// TIA Portal V16 export
// export: Created 2024-05-10T06:46:43.0449817Z, ExportSetting WithDefaults, DisplayName Totally Integrated Automation Portal, DisplayVersion V16, DisplayName TIA Portal Version Control Interface, DisplayVersion V16, DisplayName TIA Portal Openness, DisplayVersion V16, DisplayName STEP 7 Professional, DisplayVersion V16, DisplayName STEP 7 Safety, DisplayVersion V16, DisplayName WinCC Professional, DisplayVersion V16
FUNCTION_BLOCK "F120_SinaPos(SV660F)"   // FB120, LAD
{ S7_Optimized_Access := 'TRUE' }
VERSION : 0.1
// 2024/2/4:第一版本V1.0，作者:wang
// stored: AutoNumber false, IsIECCheckEnabled false, IsRetainMemResEnabled false, MemoryReserve 100, SetENOAutomatically false, UDAEnableTagReadback false
   VAR_INPUT
      IW_手动模式 { ExternalAccessible := 'False'; ExternalVisible := 'False'; ExternalWritable := 'False'} : Bool;
      IW_运行条件 { ExternalAccessible := 'False'; ExternalVisible := 'False'; ExternalWritable := 'False'} : Array[1..8] of Bool;
      IM_使能 { ExternalAccessible := 'False'; ExternalVisible := 'False'; ExternalWritable := 'False'} : Bool;
      IM_回零 { ExternalAccessible := 'False'; ExternalVisible := 'False'; ExternalWritable := 'False'} : Bool;
      IM_绝对定位 { ExternalAccessible := 'False'; ExternalVisible := 'False'; ExternalWritable := 'False'} : Bool;
      IM_相对定位 { ExternalAccessible := 'False'; ExternalVisible := 'False'; ExternalWritable := 'False'} : Bool;
      "IM_JOG+" { ExternalAccessible := 'False'; ExternalVisible := 'False'; ExternalWritable := 'False'} : Bool;
      "IM_JOG-" { ExternalAccessible := 'False'; ExternalVisible := 'False'; ExternalWritable := 'False'} : Bool;
      IM_故障复位 { ExternalAccessible := 'False'; ExternalVisible := 'False'; ExternalWritable := 'False'} : Bool;
      ID_目标位置 { ExternalAccessible := 'False'; ExternalVisible := 'False'; ExternalWritable := 'False'} : DInt;
      ID_目标速度 { ExternalAccessible := 'False'; ExternalVisible := 'False'; ExternalWritable := 'False'} : DInt;
      "IW_速度加减倍率%" { ExternalAccessible := 'False'; ExternalVisible := 'False'; ExternalWritable := 'False'} : Array[1..3] of Int;
      ID_ConfigEpos { ExternalAccessible := 'False'; ExternalVisible := 'False'; ExternalWritable := 'False'} : DWord;
      ID_111报文标识符 { ExternalAccessible := 'False'; ExternalVisible := 'False'; ExternalWritable := 'False'} : HW_IO;
   END_VAR
   VAR_OUTPUT
      OM_准备好了 : Bool;
      OM_动作中 : Bool;
      OM_回零完了 : Bool;
      OM_轴报警 : Bool;
      OM_轴错误 : Bool;
      OD_当前位置 : DInt;
      OD_当前速度 : DInt;
      OW_运行模式 : Int;
      OW_EPSW1 : Word;
      OW_EPSW2 : Word;
      OW_轴报警码 : Word;
      OW_轴错误码 : Word;
      OW_库错误码 : Int;
      OW_调用错误码 : Word;
   END_VAR
   VAR
      MT_StartChk : IEC_TIMER;   // 启动延迟
   END_VAR
   VAR_TEMP
      M_停止 : Bool;
      M_暂停 : Bool;
      M_JOG指令 : Bool;
      M_回零指令 : Bool;
      M_绝对定位指令 : Bool;
      M_相对定位指令 : Bool;
      M_回零定位完Pls : Bool;
      M_绝对定位完Pls : Bool;
      M_相对定位完Pls : Bool;
      M_启动 : Bool;
      M_定位完了 : Bool;
      W_运行模式 : Int;
      M_Pulse : Array[1..20] of Bool;
      M_SerState : Bool;   // 伺服正常
      M_Busy : Bool;   // 伺服忙
      M_FLS_SW : Bool;   // 正极限
      M_RLS_SW : Bool;   // 负极限
   END_VAR
   // // IW_运行条件[1] : 共同条件
   // // IW_运行条件[2] : 回零条件
   // // IW_运行条件[3] : JOG正条件
   // // IW_运行条件[4] : JOG负条件
   // // IW_运行条件[5] : 定位正条件
   // // IW_运行条件[6] : 定位负条件
   // // IW_运行条件[7] : 预留
   // // IW_运行条件[8] : 预留
   VAR_TEMP   // added for the SCL form of the ladder/FBD networks
      _w1 : Bool;
      _w2 : Bool;
      _w3 : Bool;
      _w4 : Bool;
   END_VAR
BEGIN

REGION Network 1: 伺服状态条件
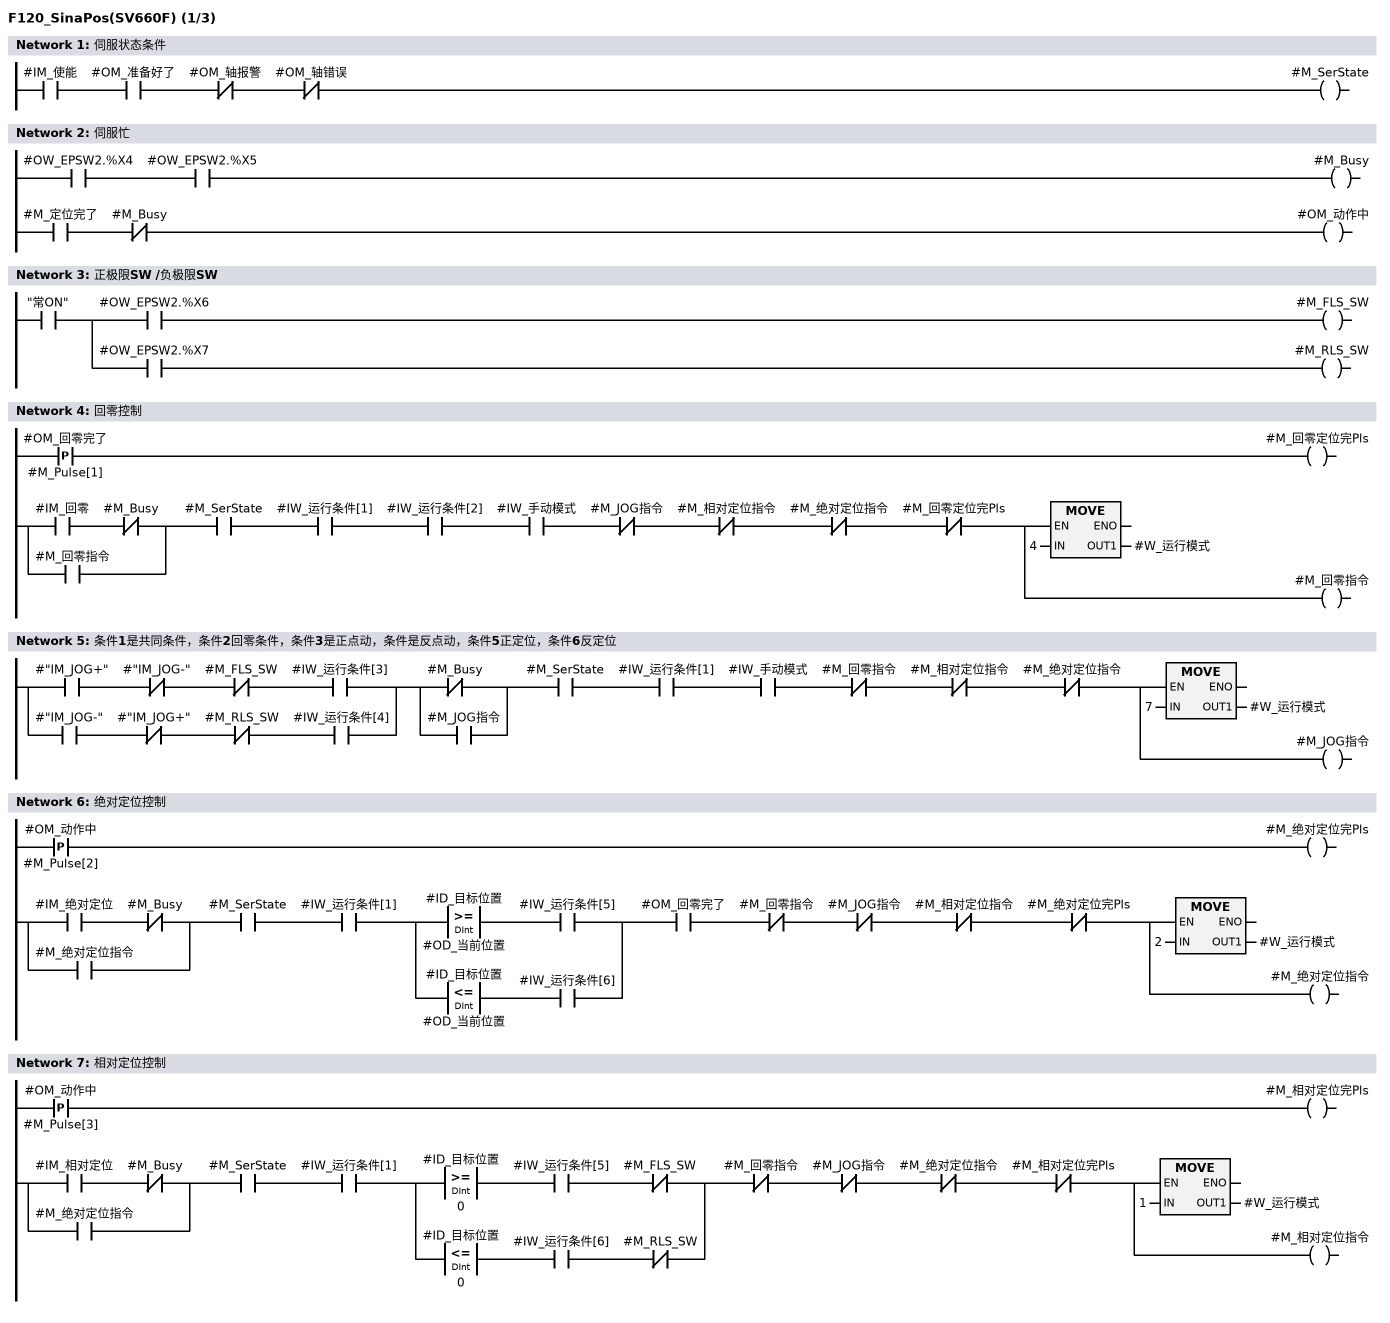
   RUNG wire#powerrail
      Contact( #IM_使能 )
      Contact( #OM_准备好了 )
      I_Contact( #OM_轴报警 )
      I_Contact( #OM_轴错误 )
      Coil( #M_SerState )
   END_RUNG
   // the same network as SCL:
   #M_SerState := #IM_使能 AND #OM_准备好了 AND NOT #OM_轴报警 AND NOT #OM_轴错误;
END_REGION

REGION Network 2: 伺服忙
   RUNG wire#powerrail
      Contact( #OW_EPSW2.%X4 )
      Contact( #OW_EPSW2.%X5 )
      Coil( #M_Busy )
   END_RUNG
   RUNG wire#powerrail
      Contact( #M_定位完了 )
      I_Contact( #M_Busy )
      Coil( #OM_动作中 )
   END_RUNG
   // the same network as SCL:
   #M_Busy := #OW_EPSW2.%X4 AND #OW_EPSW2.%X5;
   #OM_动作中 := #M_定位完了 AND NOT #M_Busy;
END_REGION

REGION Network 3: 正极限SW /负极限SW
   RUNG wire#powerrail
      Contact( "常ON" )
      wire#w1
      Contact( #OW_EPSW2.%X6 )
      Coil( #M_FLS_SW )
   END_RUNG
   RUNG wire#w1
      Contact( #OW_EPSW2.%X7 )
      Coil( #M_RLS_SW )
   END_RUNG
   // the same network as SCL:
   #M_FLS_SW := "常ON" AND #OW_EPSW2.%X6;
   #M_RLS_SW := "常ON" AND #OW_EPSW2.%X7;
END_REGION

REGION Network 4: 回零控制
   RUNG wire#powerrail
      P_Contact(operand := #OM_回零完了, bit := #M_Pulse[1])
      Coil( #M_回零定位完Pls )
   END_RUNG
   RUNG wire#powerrail
      Contact( #IM_回零 )
      I_Contact( #M_Busy )
      wire#w1
      Contact( #M_SerState )
      Contact( #IW_运行条件[1] )
      Contact( #IW_运行条件[2] )
      Contact( #IW_手动模式 )
      I_Contact( #M_JOG指令 )
      I_Contact( #M_相对定位指令 )
      I_Contact( #M_绝对定位指令 )
      I_Contact( #M_回零定位完Pls )
      wire#w2
      Move(in := 4, out1 => #W_运行模式)
   END_RUNG
   RUNG wire#powerrail
      Contact( #M_回零指令 )
   END_RUNG wire#w1
   RUNG wire#w2
      Coil( #M_回零指令 )
   END_RUNG
   // the same network as SCL:
   #_w1 := #OM_回零完了 AND NOT #M_Pulse[1];   // rising edge of #OM_回零完了
   #M_Pulse[1] := #OM_回零完了;
   #M_回零定位完Pls := #_w1;
   #_w2 := ((#IM_回零 AND NOT #M_Busy) OR #M_回零指令) AND #M_SerState AND #IW_运行条件[1] AND #IW_运行条件[2] AND #IW_手动模式 AND NOT #M_JOG指令 AND NOT #M_相对定位指令 AND NOT #M_绝对定位指令 AND NOT #M_回零定位完Pls;
   IF #_w2 THEN #W_运行模式 := 4; END_IF;
   #M_回零指令 := #_w2;
END_REGION

REGION Network 5: 条件1是共同条件，条件2回零条件，条件3是正点动，条件是反点动，条件5正定位，条件6反定位
   RUNG wire#powerrail
      Contact( #"IM_JOG+" )
      I_Contact( #"IM_JOG-" )
      I_Contact( #M_FLS_SW )
      Contact( #IW_运行条件[3] )
      wire#w1
      I_Contact( #M_Busy )
      wire#w2
      Contact( #M_SerState )
      Contact( #IW_运行条件[1] )
      Contact( #IW_手动模式 )
      I_Contact( #M_回零指令 )
      I_Contact( #M_相对定位指令 )
      I_Contact( #M_绝对定位指令 )
      wire#w3
      Move(in := 7, out1 => #W_运行模式)
   END_RUNG
   RUNG wire#powerrail
      Contact( #"IM_JOG-" )
      I_Contact( #"IM_JOG+" )
      I_Contact( #M_RLS_SW )
      Contact( #IW_运行条件[4] )
   END_RUNG wire#w1
   RUNG wire#w1
      Contact( #M_JOG指令 )
   END_RUNG wire#w2
   RUNG wire#w3
      Coil( #M_JOG指令 )
   END_RUNG
   // the same network as SCL:
   #_w1 := ((#"IM_JOG+" AND NOT #"IM_JOG-" AND NOT #M_FLS_SW AND #IW_运行条件[3]) OR (#"IM_JOG-" AND NOT #"IM_JOG+" AND NOT #M_RLS_SW AND #IW_运行条件[4])) AND (NOT #M_Busy OR #M_JOG指令) AND #M_SerState AND #IW_运行条件[1] AND #IW_手动模式 AND NOT #M_回零指令 AND NOT #M_相对定位指令 AND NOT #M_绝对定位指令;
   IF #_w1 THEN #W_运行模式 := 7; END_IF;
   #M_JOG指令 := #_w1;
END_REGION

REGION Network 6: 绝对定位控制
   RUNG wire#powerrail
      P_Contact(operand := #OM_动作中, bit := #M_Pulse[2])
      Coil( #M_绝对定位完Pls )
   END_RUNG
   RUNG wire#powerrail
      Contact( #IM_绝对定位 )
      I_Contact( #M_Busy )
      wire#w1
      Contact( #M_SerState )
      Contact( #IW_运行条件[1] )
      wire#w2
      { S7_Templates := "SrcType := DInt" } GE_Contact(in1 := #ID_目标位置, in2 := #OD_当前位置)
      Contact( #IW_运行条件[5] )
      wire#w3
      Contact( #OM_回零完了 )
      I_Contact( #M_回零指令 )
      I_Contact( #M_JOG指令 )
      I_Contact( #M_相对定位指令 )
      I_Contact( #M_绝对定位完Pls )
      wire#w4
      Move(in := 2, out1 => #W_运行模式)
   END_RUNG
   RUNG wire#powerrail
      Contact( #M_绝对定位指令 )
   END_RUNG wire#w1
   RUNG wire#w2
      { S7_Templates := "SrcType := DInt" } LE_Contact(in1 := #ID_目标位置, in2 := #OD_当前位置)
      Contact( #IW_运行条件[6] )
   END_RUNG wire#w3
   RUNG wire#w4
      Coil( #M_绝对定位指令 )
   END_RUNG
   // the same network as SCL:
   #_w1 := #OM_动作中 AND NOT #M_Pulse[2];   // rising edge of #OM_动作中
   #M_Pulse[2] := #OM_动作中;
   #M_绝对定位完Pls := #_w1;
   #_w2 := ((#IM_绝对定位 AND NOT #M_Busy) OR #M_绝对定位指令) AND #M_SerState AND #IW_运行条件[1] AND (((#ID_目标位置 >= #OD_当前位置) AND #IW_运行条件[5]) OR ((#ID_目标位置 <= #OD_当前位置) AND #IW_运行条件[6])) AND #OM_回零完了 AND NOT #M_回零指令 AND NOT #M_JOG指令 AND NOT #M_相对定位指令 AND NOT #M_绝对定位完Pls;
   IF #_w2 THEN #W_运行模式 := 2; END_IF;
   #M_绝对定位指令 := #_w2;
END_REGION

REGION Network 7: 相对定位控制
   RUNG wire#powerrail
      P_Contact(operand := #OM_动作中, bit := #M_Pulse[3])
      Coil( #M_相对定位完Pls )
   END_RUNG
   RUNG wire#powerrail
      Contact( #IM_相对定位 )
      I_Contact( #M_Busy )
      wire#w1
      Contact( #M_SerState )
      Contact( #IW_运行条件[1] )
      wire#w2
      { S7_Templates := "SrcType := DInt" } GE_Contact(in1 := #ID_目标位置, in2 := 0)
      Contact( #IW_运行条件[5] )
      I_Contact( #M_FLS_SW )
      wire#w3
      I_Contact( #M_回零指令 )
      I_Contact( #M_JOG指令 )
      I_Contact( #M_绝对定位指令 )
      I_Contact( #M_相对定位完Pls )
      wire#w4
      Move(in := 1, out1 => #W_运行模式)
   END_RUNG
   RUNG wire#powerrail
      Contact( #M_绝对定位指令 )
   END_RUNG wire#w1
   RUNG wire#w2
      { S7_Templates := "SrcType := DInt" } LE_Contact(in1 := #ID_目标位置, in2 := 0)
      Contact( #IW_运行条件[6] )
      I_Contact( #M_RLS_SW )
   END_RUNG wire#w3
   RUNG wire#w4
      Coil( #M_相对定位指令 )
   END_RUNG
   // the same network as SCL:
   #_w1 := #OM_动作中 AND NOT #M_Pulse[3];   // rising edge of #OM_动作中
   #M_Pulse[3] := #OM_动作中;
   #M_相对定位完Pls := #_w1;
   #_w2 := ((#IM_相对定位 AND NOT #M_Busy) OR #M_绝对定位指令) AND #M_SerState AND #IW_运行条件[1] AND (((#ID_目标位置 >= 0) AND #IW_运行条件[5] AND NOT #M_FLS_SW) OR ((#ID_目标位置 <= 0) AND #IW_运行条件[6] AND NOT #M_RLS_SW)) AND NOT #M_回零指令 AND NOT #M_JOG指令 AND NOT #M_绝对定位指令 AND NOT #M_相对定位完Pls;
   IF #_w2 THEN #W_运行模式 := 1; END_IF;
   #M_相对定位指令 := #_w2;
END_REGION

REGION Network 8: 控制启动
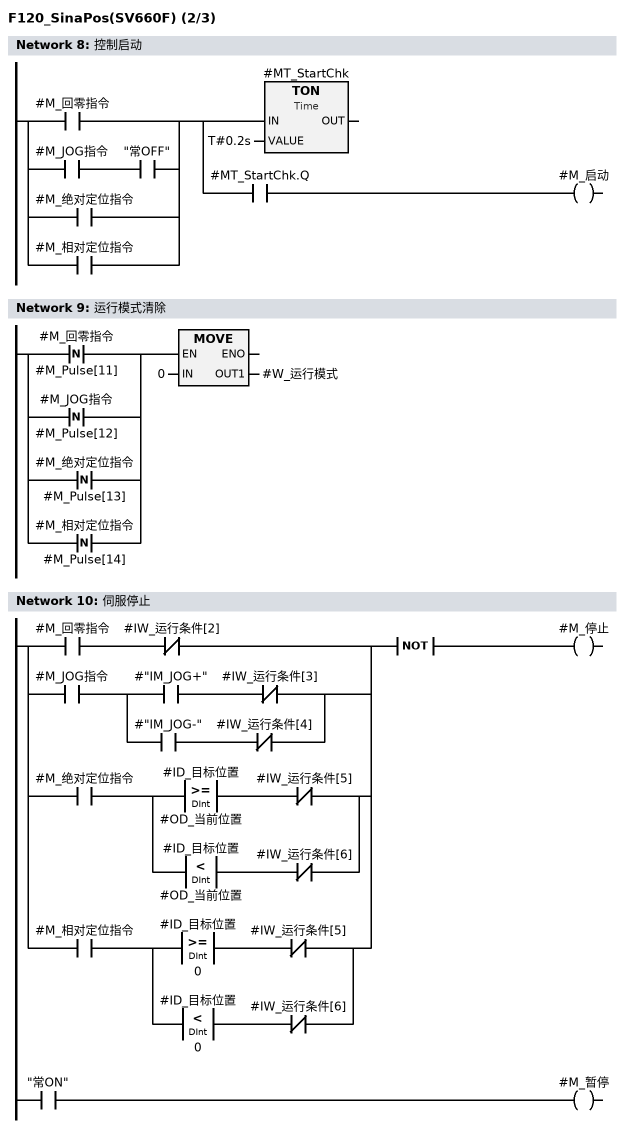
   #_w1 := #M_回零指令 OR (#M_JOG指令 AND "常OFF") OR #M_绝对定位指令 OR #M_相对定位指令;
   #MT_StartChk.TON(IN := #_w1, PT := T#0.2s);   // TON coil
   #M_启动 := #_w1 AND #MT_StartChk.Q;
END_REGION

REGION Network 9: 运行模式清除
   RUNG wire#powerrail
      N_Contact(operand := #M_回零指令, bit := #M_Pulse[11])
      wire#w1
      Move(in := 0, out1 => #W_运行模式)
   END_RUNG
   RUNG wire#powerrail
      N_Contact(operand := #M_JOG指令, bit := #M_Pulse[12])
   END_RUNG wire#w1
   RUNG wire#powerrail
      N_Contact(operand := #M_绝对定位指令, bit := #M_Pulse[13])
   END_RUNG wire#w1
   RUNG wire#powerrail
      N_Contact(operand := #M_相对定位指令, bit := #M_Pulse[14])
   END_RUNG wire#w1
   // the same network as SCL:
   #_w1 := NOT #M_回零指令 AND #M_Pulse[11];   // falling edge of #M_回零指令
   #M_Pulse[11] := #M_回零指令;
   #_w2 := NOT #M_JOG指令 AND #M_Pulse[12];   // falling edge of #M_JOG指令
   #M_Pulse[12] := #M_JOG指令;
   #_w3 := NOT #M_绝对定位指令 AND #M_Pulse[13];   // falling edge of #M_绝对定位指令
   #M_Pulse[13] := #M_绝对定位指令;
   #_w4 := NOT #M_相对定位指令 AND #M_Pulse[14];   // falling edge of #M_相对定位指令
   #M_Pulse[14] := #M_相对定位指令;
   IF #_w1 OR #_w2 OR #_w3 OR #_w4 THEN #W_运行模式 := 0; END_IF;
END_REGION

REGION Network 10: 伺服停止
   RUNG wire#powerrail
      Contact( #M_回零指令 )
      I_Contact( #IW_运行条件[2] )
      wire#w1
      Not()
      Coil( #M_停止 )
   END_RUNG
   RUNG wire#powerrail
      Contact( #M_JOG指令 )
      wire#w2
      Contact( #"IM_JOG+" )
      I_Contact( #IW_运行条件[3] )
   END_RUNG wire#w1
   RUNG wire#w2
      Contact( #"IM_JOG-" )
      I_Contact( #IW_运行条件[4] )
   END_RUNG wire#w1
   RUNG wire#powerrail
      Contact( #M_绝对定位指令 )
      wire#w3
      { S7_Templates := "SrcType := DInt" } GE_Contact(in1 := #ID_目标位置, in2 := #OD_当前位置)
      I_Contact( #IW_运行条件[5] )
   END_RUNG wire#w1
   RUNG wire#w3
      { S7_Templates := "SrcType := DInt" } LT_Contact(in1 := #ID_目标位置, in2 := #OD_当前位置)
      I_Contact( #IW_运行条件[6] )
   END_RUNG wire#w1
   RUNG wire#powerrail
      Contact( #M_相对定位指令 )
      wire#w4
      { S7_Templates := "SrcType := DInt" } GE_Contact(in1 := #ID_目标位置, in2 := 0)
      I_Contact( #IW_运行条件[5] )
   END_RUNG wire#w1
   RUNG wire#w4
      { S7_Templates := "SrcType := DInt" } LT_Contact(in1 := #ID_目标位置, in2 := 0)
      I_Contact( #IW_运行条件[6] )
   END_RUNG wire#w1
   RUNG wire#powerrail
      Contact( "常ON" )
      Coil( #M_暂停 )
   END_RUNG
   // the same network as SCL:
   #M_停止 := NOT ((#M_回零指令 AND NOT #IW_运行条件[2]) OR (#M_JOG指令 AND ((#"IM_JOG+" AND NOT #IW_运行条件[3]) OR (#"IM_JOG-" AND NOT #IW_运行条件[4]))) OR (#M_绝对定位指令 AND (((#ID_目标位置 >= #OD_当前位置) AND NOT #IW_运行条件[5]) OR ((#ID_目标位置 < #OD_当前位置) AND NOT #IW_运行条件[6]))) OR (#M_相对定位指令 AND (((#ID_目标位置 >= 0) AND NOT #IW_运行条件[5]) OR ((#ID_目标位置 < 0) AND NOT #IW_运行条件[6]))));
   #M_暂停 := "常ON";
END_REGION

REGION Network 11
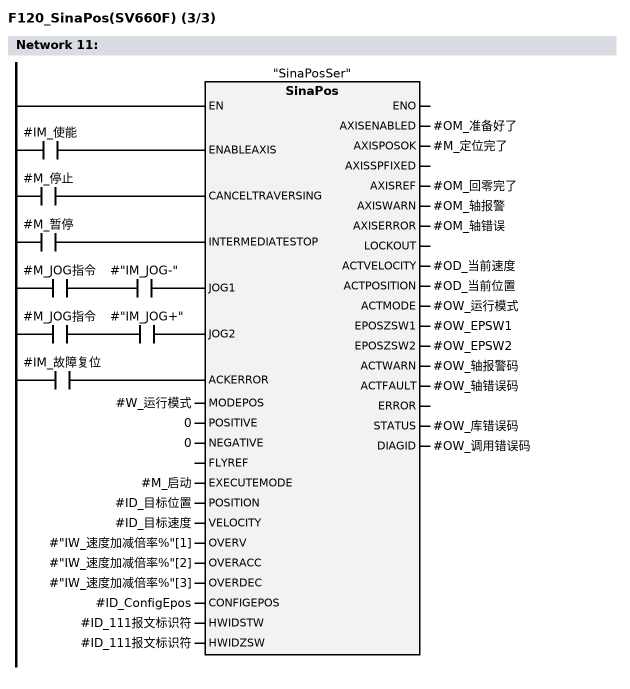
   RUNG wire#powerrail
      "SinaPosSer".SinaPos(EnableAxis := wire#w1, CancelTraversing := wire#w2, IntermediateStop := wire#w3, Jog1 := wire#w4, Jog2 := wire#w5, AckError := wire#w6, ModePos := #W_运行模式, Positive := 0, Negative := 0, FlyRef :=, ExecuteMode := #M_启动, Position := #ID_目标位置, Velocity := #ID_目标速度, OverV := #"IW_速度加减倍率%"[1], OverAcc := #"IW_速度加减倍率%"[2], OverDec := #"IW_速度加减倍率%"[3], ConfigEPos := #ID_ConfigEpos, HWIDSTW := #ID_111报文标识符, HWIDZSW := #ID_111报文标识符, AxisEnabled => #OM_准备好了, AxisPosOk => #M_定位完了, AxisSpFixed =>, AxisRef => #OM_回零完了, AxisWarn => #OM_轴报警, AxisError => #OM_轴错误, Lockout =>, ActVelocity => #OD_当前速度, ActPosition => #OD_当前位置, ActMode => #OW_运行模式, EPosZSW1 => #OW_EPSW1, EPosZSW2 => #OW_EPSW2, ActWarn => #OW_轴报警码, ActFault => #OW_轴错误码, Error =>, Status => #OW_库错误码, DiagId => #OW_调用错误码)
   END_RUNG
   RUNG wire#powerrail
      Contact( #IM_使能 )
   END_RUNG wire#w1
   RUNG wire#powerrail
      Contact( #M_停止 )
   END_RUNG wire#w2
   RUNG wire#powerrail
      Contact( #M_暂停 )
   END_RUNG wire#w3
   RUNG wire#powerrail
      Contact( #M_JOG指令 )
      Contact( #"IM_JOG-" )
   END_RUNG wire#w4
   RUNG wire#powerrail
      Contact( #M_JOG指令 )
      Contact( #"IM_JOG+" )
   END_RUNG wire#w5
   RUNG wire#powerrail
      Contact( #IM_故障复位 )
   END_RUNG wire#w6
   // the same network as SCL:
   "SinaPosSer"(EnableAxis := #IM_使能,   // SinaPos
                CancelTraversing := #M_停止,
                IntermediateStop := #M_暂停,
                Jog1 := #M_JOG指令 AND #"IM_JOG-",
                Jog2 := #M_JOG指令 AND #"IM_JOG+",
                AckError := #IM_故障复位,
                ModePos := #W_运行模式,
                Positive := 0,
                Negative := 0,
                ExecuteMode := #M_启动,
                Position := #ID_目标位置,
                Velocity := #ID_目标速度,
                OverV := #"IW_速度加减倍率%"[1],
                OverAcc := #"IW_速度加减倍率%"[2],
                OverDec := #"IW_速度加减倍率%"[3],
                ConfigEPos := #ID_ConfigEpos,
                HWIDSTW := #ID_111报文标识符,
                HWIDZSW := #ID_111报文标识符,
                AxisEnabled => #OM_准备好了,
                AxisPosOk => #M_定位完了,
                AxisRef => #OM_回零完了,
                AxisWarn => #OM_轴报警,
                AxisError => #OM_轴错误,
                ActVelocity => #OD_当前速度,
                ActPosition => #OD_当前位置,
                ActMode => #OW_运行模式,
                EPosZSW1 => #OW_EPSW1,
                EPosZSW2 => #OW_EPSW2,
                ActWarn => #OW_轴报警码,
                ActFault => #OW_轴错误码,
                Status => #OW_库错误码,
                DiagId => #OW_调用错误码);
END_REGION
END_FUNCTION_BLOCK
